TYPE ST_SensorDataSets :
STRUCT
	sName			: STRING;
	sPlcName		: STRING;
	stFieldPoints	: ARRAY[1..MAX_NO_OF_FIELD_POINT] OF ST_FieldPoint; 	
END_STRUCT
END_TYPE

(* stored: Version 1.1.0.1, ProductVersion 3.1.4024.4
   DUT ST_SensorDataSets: Id {5403556c-5c31-4efb-90f8-ab256c41686d} *)
